FUNCTION_BLOCK FB_WriteLimits
VAR_INPUT
	bExecute	: BOOL;
	dnUpLimit	: DINT;
	dnDownLimit	: DINT;
END_VAR
VAR_OUTPUT
	
	bDone 		: BOOL;	//both limits were written and verified
	bError		: BOOL; //Error writing or limits not verified
	udnErrorID	: UDINT;	//Error code, to be added to later (writing or reading)
	bBusy		: BOOL;	//in the process of running the Function Blocks

	
END_VAR
VAR
	fbMC_WriteUPParameter: MC_WriteParameter;
	fbMc_WriteDownParameter: MC_WriteParameter;
	WriteLimits: INT;
	fbMC_ReadUPParameter: MC_ReadParameter;
	fbMC_ReadDownParameter: MC_ReadParameter;
END_VAR
VAR_IN_OUT
	Axis		: Axis_Ref;
	
END_VAR

	
CASE WriteLimits OF
	
	0 :	//wait for the bExecute
		IF bExecute THEN
			bError		:= FALSE;
			udnErrorID	:= 0;
			bBusy		:= TRUE;
			WriteLimits := 2;
		END_IF

	2 :	//setting Function Block to False
		fbMC_WriteUPParameter(Axis:= Axis ,Execute:= FALSE);
		WriteLimits := WriteLimits +1;	
		
	3 :	//write to the up limit	
		
		fbMC_WriteUPParameter(		//Execute the Write Parameter for NC
			Axis			:= Axis ,
			Execute			:= TRUE, 
			ParameterNumber	:= AxisMaxSoftPosLimit, 
			Value			:= DINT_TO_LREAL(dnUpLimit), 
			Done			=> , 
			Busy			=> , 
			Error			=> , 
			ErrorID			=> udnErrorID);
		
		IF fbMC_WriteUPParameter.Error THEN
			
			WriteLimits := 9999;
			//Add error handling 
		ELSE
			IF fbMC_WriteUPParameter.Done THEN
				fbMC_WriteUPParameter(Axis:= Axis ,Execute:= FALSE);
				WriteLimits := WriteLimits +1;
			END_IF
		END_IF	
		
	4:	//Setting FB to False
		fbMC_ReadUPParameter(Axis:= Axis ,Enable:= FALSE);
		WriteLimits := WriteLimits +1;	
	
	5:	//Reading last value of UpLimit written in Case 4
		fbMC_ReadUPParameter(
			Axis:= Axis, 
			Enable:= TRUE, 
			ParameterNumber:= AxisMaxSoftPosLimit, 
			ReadMode:= ReadMode_Once, 
			Valid=> , 
			Busy=> , 
			Error=> , 
			ErrorID=> , 
			Value=> );

		IF fbMC_ReadUPParameter.Error THEN
			WriteLimits := 9999;
			//Add error handling 
		ELSE
			IF NOT fbMC_ReadUPParameter.Busy THEN
				fbMC_ReadUPParameter(Axis:= Axis ,Enable:= FALSE);
				WriteLimits := WriteLimits +1;
			END_IF
		END_IF		
			
	6:	//Comparison of Written Value to Read Value
	
		IF fbMC_ReadUPParameter.Value = DINT_TO_LREAL(dnUpLimit) THEN
			WriteLimits := WriteLimits +1;
		ELSE
			WriteLimits := 9999;
		END_IF
		
	7:	//setting Function Block to False
		fbMC_WriteDownParameter(Axis:= Axis ,Execute:= FALSE);
		WriteLimits := WriteLimits +1;	
		
	8 :	//write to the down limit	
		
		fbMC_WriteDownParameter(		//Execute the Write Parameter for NC
			Axis			:= Axis ,
			Execute			:= TRUE, 
			ParameterNumber	:= AxisMinSoftPosLimit, 
			Value			:= DINT_TO_LREAL(dnDownLimit), 
			Done			=> , 
			Busy			=> , 
			Error			=> , 
			ErrorID			=> udnErrorID);
		
		IF fbMC_WriteDownParameter.Error THEN
			
			WriteLimits := 9999;
			//Add error handling 
		ELSE
			IF fbMC_WriteDownParameter.Done THEN
				fbMC_WriteDownParameter(Axis:= Axis ,Execute:= FALSE);
				WriteLimits := WriteLimits +1;
			END_IF
		END_IF	
		
	9:	//Setting FB to False
		fbMC_ReadDownParameter(Axis:= Axis ,Enable:= FALSE);
		WriteLimits := WriteLimits +1;	
	
	10:	//Reading last value of UpLimit written in Case 4
		fbMC_ReadDownParameter(
			Axis:= Axis, 
			Enable:= TRUE, 
			ParameterNumber:= AxisMinSoftPosLimit, 
			ReadMode:= ReadMode_Once, 
			Valid=> , 
			Busy=> , 
			Error=> , 
			ErrorID=> , 
			Value=> );

		IF fbMC_ReadDownParameter.Error THEN
			WriteLimits := 9999;
			//Add error handling 
		ELSE
			IF NOT fbMC_ReadDownParameter.Busy THEN
				fbMC_ReadDownParameter(Axis:= Axis ,Enable:= FALSE);
				WriteLimits := WriteLimits +1;
			END_IF
		END_IF		
			
	11:	//Comparison of Written Value to Read Value
	
		IF fbMC_ReadDownParameter.Value = DINT_TO_LREAL(dnDownLimit) THEN
			fbMC_WriteUPParameter(Axis := Axis, Execute := FALSE);
			WriteLimits := WriteLimits +1;
		ELSE
			WriteLimits := 9999;
		END_IF
	
	12: //Verify that Soft Limit Switch is enabled
	
	fbMC_WriteUPParameter(		//Execute the Write Parameter for NC
			Axis			:= Axis ,
			Execute			:= TRUE, 
			ParameterNumber	:= AxisEnMaxSoftPosLimit, 
			Value			:= BOOL_TO_LREAL(TRUE), 
			Done			=> , 
			Busy			=> , 
			Error			=> , 
			ErrorID			=> udnErrorID);
		
		IF fbMC_WriteUPParameter.Error THEN
			
			WriteLimits := 9999;
			//Add error handling 
		ELSE
			IF fbMC_WriteUPParameter.Done THEN
				fbMC_WriteUPParameter(Axis:= Axis ,Execute:= FALSE);
				WriteLimits := WriteLimits +1;
			END_IF
		END_IF	
		
	13:	//Setting FB to False
		fbMC_ReadUPParameter(Axis:= Axis ,Enable:= FALSE);
		WriteLimits := WriteLimits +1;	
	
	14:	//Reading last value of UpLimit written in Case 4
		fbMC_ReadUPParameter(
			Axis:= Axis, 
			Enable:= TRUE, 
			ParameterNumber:= AxisEnMaxSoftPosLimit, 
			ReadMode:= ReadMode_Once, 
			Valid=> , 
			Busy=> , 
			Error=> , 
			ErrorID=> , 
			Value=> );

		IF fbMC_ReadUPParameter.Error THEN
			WriteLimits := 9999;
			//Add error handling 
		ELSE
			IF NOT fbMC_ReadUPParameter.Busy THEN
				fbMC_ReadUPParameter(Axis:= Axis ,Enable:= FALSE);
				WriteLimits := WriteLimits +1;
			END_IF
		END_IF		
			
	15:	//Comparison of Written Value to Read Value
	
		IF fbMC_ReadUPParameter.Value = BOOL_TO_LREAL(TRUE) THEN
			WriteLimits := WriteLimits +1;
		ELSE
			WriteLimits := 9999;
		END_IF
		
	16:	//setting Function Block to False
		fbMC_WriteDownParameter(Axis:= Axis ,Execute:= FALSE);
		WriteLimits := WriteLimits +1;
		
	17:	//write to the down limit	
		
		fbMC_WriteDownParameter(		//Execute the Write Parameter for NC
			Axis			:= Axis ,
			Execute			:= TRUE, 
			ParameterNumber	:= AxisEnMinSoftPosLimit, 
			Value			:= BOOL_TO_LREAL(TRUE), 
			Done			=> , 
			Busy			=> , 
			Error			=> , 
			ErrorID			=> udnErrorID);
		
		IF fbMC_WriteDownParameter.Error THEN
			
			WriteLimits := 9999;
			//Add error handling 
		ELSE
			IF fbMC_WriteDownParameter.Done THEN
				fbMC_WriteDownParameter(Axis:= Axis ,Execute:= FALSE);
				WriteLimits := WriteLimits +1;
			END_IF
		END_IF	
		
	18:	//Setting FB to False
		fbMC_ReadDownParameter(Axis:= Axis ,Enable:= FALSE);
		WriteLimits := WriteLimits +1;
	
	19:	//Reading last value of UpLimit written in Case 4
		fbMC_ReadDownParameter(
			Axis:= Axis, 
			Enable:= TRUE, 
			ParameterNumber:= AxisEnMinSoftPosLimit, 
			ReadMode:= ReadMode_Once, 
			Valid=> , 
			Busy=> , 
			Error=> , 
			ErrorID=> , 
			Value=> );

		IF fbMC_ReadDownParameter.Error THEN
			WriteLimits := 9999;
			//Add error handling 
		ELSE
			IF NOT fbMC_ReadDownParameter.Busy THEN
				fbMC_ReadDownParameter(Axis:= Axis ,Enable:= FALSE);
				WriteLimits := WriteLimits +1;
			END_IF
		END_IF		
			
	20:	//Comparison of Written Value to Read Value
	
		IF fbMC_ReadDownParameter.Value = BOOL_TO_LREAL(TRUE) THEN
			WriteLimits := 10000;
		ELSE
			WriteLimits := 9999;
		END_IF

	
	9999:	//Error Handling
		bError  := TRUE;
		bBusy	:= FALSE;
				
		IF NOT bExecute THEN
			WriteLimits := 0;
		END_IF	
	
	10000:	//Done writing and verifying limits
		bBusy	:= FALSE;
		bDone	:= TRUE;
		
		IF NOT bExecute THEN
			WriteLimits := 0;
			bDone		:= false;
		END_IF	
		
END_CASE

END_FUNCTION_BLOCK

(* stored: Version 1.1.0.1, ProductVersion 3.1.4022.3
   POU FB_WriteLimits: Id {c9e7c7b0-63fe-47fd-92fc-57e8720fad07}, SpecialFunc None *)
